// TwinCAT 3 PLC project LSS_LIB
// Title: LSS
// Company: SLAC
// ProjectVersion: 0.0.0
// ProgramVersion: 3.1.4026.17
// libraries:
//   Tc2_SerialCom, * (Beckhoff Automation GmbH)
//   Tc2_Standard, * (Beckhoff Automation GmbH)
//   Tc2_System, * (Beckhoff Automation GmbH)
//   Tc2_Utilities, * (Beckhoff Automation GmbH)
// project tree:
//   DUTs/ E_ALPHA_LED_LINE_POSITION.TcDUT, E_ALPHA_MULTIPLEX_ITEM.TcDUT
//   / PlcTask.TcTTO
//   POUs/ FB_Alpha215C.TcPOU, FB_ALPHA215C_Multiplex.TcPOU, MAIN.TcPOU
// real-time tasks:
//   TASK PlcTask: cycle T#10ms, priority 20, ADS port 350

CONFIGURATION LSS_LIB
    RESOURCE PLC ON TwinCAT3
        TASK PlcTask(INTERVAL := T#10ms, PRIORITY := 20);
        PROGRAM MAIN WITH PlcTask : MAIN;
    END_RESOURCE
END_CONFIGURATION

// ---- DUTs/E_ALPHA_LED_LINE_POSITION.TcDUT
{attribute 'qualified_only'}
{attribute 'strict'}
{attribute 'to_string'}
TYPE E_ALPHA_LED_LINE_POSITION :
(
    MIDDLE_LINE := 0 	// — Text centered vertically
    (*
    TOP_LINE, 			(*— Text begins on the top line of the sign and the sign will use all its lines minus 1 in order
                        to display the text. For example, a 6-line sign will allow a maximum of 5 lines (6 minus 1) for the Top
                        Position. The Top/Bottom Line break will remain fixed until the next Middle or Fill position is
                        specified*)
    BOTTOM_LINE, 		(* — The starting position of the Bottom Line(s) immediately follows the last line of the
                        Top Line. For example, a 6-line sign with 3 lines of text associated with the Top Line would start the
                        Bottom Line text on the 4th line of the sign. *)

    FILL				(*he sign will fill all available lines, centering the lines vertically*)
    *)
);
END_TYPE

// ---- DUTs/E_ALPHA_MULTIPLEX_ITEM.TcDUT
TYPE E_ALPHA_MULTIPLEX_ITEM :
STRUCT
    sMessage : STRING := ' ';
    sAddress : STRING := '00'; // Display on all signs. Or Specific
    sFile	: STRING := '0'; // Sign Default configuration file 1; file 0 is priotiry
    tTime : TIME := T#1S; // How long message should display
    bActive : BOOL := FALSE; // Message should be displayed.
END_STRUCT
END_TYPE

// ---- POUs/MAIN.TcPOU
PROGRAM MAIN
VAR
END_VAR

END_PROGRAM

// ---- POUs/FB_Alpha215C.TcPOU
FUNCTION_BLOCK FB_Alpha215C
(*This FB can be used to send print commands to the ALpha Signs*)
VAR_INPUT
END_VAR
VAR_OUTPUT
END_VAR
VAR
	fbBackgroundSerialLine: SerialLineControl;
	RxBuffer:   ComBuffer;
    TxBuffer:   ComBuffer;

	// Link to hardware.
	stComIn		AT %I*	:	EL6inData22B (*KL6inData22B*);
    stComOut	AT %Q*	:	EL6outData22B (*KL6outData22B*);

	//sCommand : STRING := '';  // (sCommand = sCommandCode + sDataField) + sCommand // NESTING commands
	//sSendMessage : STRING := '_00_00_00_00_00_01Z00_02A0_1Ba_1A9_1C1NO ACCESS_04';

	bBackgroundComError: BOOL;
	bBackgroundErrorId: UINT;
	bBackgroundTaskRunning : BOOL;

	fbClearComBuffer		: ClearComBuffer;
    fbSendString			: SendString;
    fbReceiveString			: ReceiveString;

	sSendPacket : STRING := '';

	bExecuteSend : BOOL := FALSE;
	iState : UINT := 0;

	fbRingBuff : FB_StringRingBuffer;
	fbBufferMemory    : ARRAY[0..2048] OF BYTE;
	
	tTimer : TON;

END_VAR

fbRingBuff(pBuffer := ADR(fbBufferMemory), cbBuffer := SIZEOF(fbBufferMemory));
tTimer(IN:=TRUE, PT:= T#100MS);

CASE iState OF
	0:
		IF bExecuteSend THEN // Manual Send
			fbSendString.SendString := sSendPacket;
			fbClearComBuffer(Buffer:=TxBuffer);
			iState := 10;
		END_IF

		IF fbRingBuff.nCount > 0 THEN // Send w/ ring buffer
			fbRingBuff.A_RemoveHead();
			sSendPacket := fbRingBuff.getValue;
			fbSendString.SendString := sSendPacket;
			fbClearComBuffer(Buffer:=TxBuffer);
			iState := 10;
		END_IF

	10: // SEND PACKET

		fbSendString(TXbuffer:=TxBuffer);

		IF NOT fbSendString.Busy AND fbSendString.Error = 0 THEN
			tTimer.IN := FALSE;
			tTimer();
			iState := 20;
		END_IF
		
	20: // WAIT FOR NEXT MESSAGE TO SEND
		IF tTimer.Q THEN
			bExecuteSend := FALSE;
			sSendPacket := '';
			iState := 0;
		END_IF

END_CASE

ACTION A_RUN_BACKGROUND_SERIAL_CONTROL:

bBackgroundTaskRunning := TRUE;

fbBackgroundSerialLine(
	Mode := ComSerialLineMode_t.SERIALLINEMODE_EL6_22B,
	pComIn := ADR(stComIn),
	pComOut := ADR(stComout),
	SizeComIn:= UINT_TO_INT(SIZEOF(stComout)),
    TxBuffer:= TxBuffer,
    RxBuffer:= RxBuffer,
	Error => bBackgroundComError,
	ErrorID => bBackgroundErrorId);
END_ACTION

METHOD PRIVATE M_BUILD_PACKET : STRING
VAR_INPUT
	sCommand : STRING;
	sAddress : STRING;
END_VAR
VAR
	sPacket : STRING := '';
	// TRANSMISSION FORMAT: <NULL> <SOH> <TypeCode> <SignAdress> <STX> <CommandCode> <DataField> <EOT>

	NULL : STRING := '_00_00_00_00_00';	(*A minimum of five <NUL>s (00H) must be transmitted as packet synchronization characters.
											 Five <SOH>s (01H) may be substituted for the five <NUL>s.
											 The sign uses these five characters to establish the baud rate *)

	SOH : STRING := '_01';	// Start of Header
	TYPE_CODE : STRING := 'Z';	// Set Type of Sign; 'Z' = All signs
	STX : STRING :='_02'; 		//“Start of TeXt” (02H) character. <STX> always precedes a Command Code.
	EOT : STRING:= '_04';		// "End of Transmission'
END_VAR
sPacket := CONCAT(sPacket, NULL);
sPacket := CONCAT(sPacket, SOH);
sPacket := CONCAT(sPacket, TYPE_CODE);
sPacket := CONCAT(sPacket, sAddress);
sPacket := CONCAT(sPacket, STX);
sPacket := CONCAT(sPacket, sCommand);
sPacket := CONCAT(sPacket, EOT);

M_BUILD_PACKET := sPacket;
END_METHOD

METHOD PRIVATE M_BUILD_TEXT_WRITE_COMMAND : STRING
VAR_INPUT
	sMessage : STRING;
	iFile : STRING := '0'; // print to priotiry file; so message shows up immediatly
	eLinePos : E_ALPHA_LED_LINE_POSITION := E_ALPHA_LED_LINE_POSITION.MIDDLE_LINE;

END_VAR
VAR
	COMMAND_CODE : STRING := 'A'; // A = WRITE TO 'FILE'
	ESC : STRING := '_1B';
	LINE_POS : STRING;
	MODE_CODE : STRING := 'b_1C1'; // func that chains multiple codes? ; Holds Text in place (b); red color text (_1C1) - this can chain multiple codes.
	SPECIAL_MODE : STRING := ''; // CAN ALSO BE ENUM
	// A - WRITE
	// 0 - FILE LABEL ;0 is Prority
	// _1B - ESCAPE CHAR
	// '' - LINE POSITION
	// a - MODE CODE
	// '' - SPECIAL MODE
	// _1A9_1C1NO ACCESS - TEXT

	sCommand : STRING;
END_VAR
CASE eLinePos OF
	E_ALPHA_LED_LINE_POSITION.MIDDLE_LINE:
		LINE_POS := ' ';
END_CASE

sCommand := CONCAT(sCommand, COMMAND_CODE);
sCommand := CONCAT(sCommand, iFile);
sCommand := CONCAT(sCommand, ESC);
sCommand := CONCAT(sCommand, LINE_POS);
sCommand := CONCAT(sCommand, MODE_CODE);
sCommand := CONCAT(sCommand, SPECIAL_MODE);
sCommand := CONCAT(sCommand, sMessage);

M_BUILD_TEXT_WRITE_COMMAND := sCommand;
END_METHOD

METHOD M_Print : BOOL
VAR_INPUT
	sAddress : STRING := '00'; // default broadcast to all
	iFile : STRING := '0'; // Use Priority file to instantly send message to sign.
	sMessage : STRING;
END_VAR
VAR
	sCommand : STRING;
	sPacket : STRING;
END_VAR
sCommand := M_BUILD_TEXT_WRITE_COMMAND(sMessage, iFile);
sPacket := M_BUILD_PACKET(sCommand, sAddress);

fbRingBuff.putValue := sPacket;
fbRingBuff.A_AddTail();
END_METHOD

END_FUNCTION_BLOCK

// ---- POUs/FB_ALPHA215C_Multiplex.TcPOU
FUNCTION_BLOCK FB_ALPHA215C_Multiplex
(*This FB Add Messages to sign and cycle though multiple messages. Idealy One FB per Sign.
Otherwise some messages will display longer in some signs.

st_message
- message 	(string)
- duration	(time)

*)
VAR_INPUT
END_VAR
VAR_IN_OUT
    aMessages : ARRAY [*] OF E_ALPHA_MULTIPLEX_ITEM;
    aAlphaDriver : FB_Alpha215C;
END_VAR
VAR
    iCurrentItem : DINT :=  LOWER_BOUND(aMessages,1);
    iMultiplexState : UINT := 10;
    tTimer : TON;
    stItem : E_ALPHA_MULTIPLEX_ITEM;

END_VAR

tTimer(IN:=TRUE);

CASE iMultiplexState OF
    10: // START PRINTING
        stItem := aMessages[iCurrentItem];

        IF stItem.bActive THEN
            aAlphaDriver.M_Print(sAddress := stItem.sAddress,
                iFile := stItem.sFile,
                sMessage := stItem.sMessage
            );

            tTimer.PT := stItem.tTime;
        ELSE
            tTimer.PT := T#0S;
        END_IF

        tTimer.IN := FALSE; // START TIMER
        tTimer();
        iMultiplexState := 20;

    20: // Wait
        IF tTimer.Q THEN //
            iCurrentItem := iCurrentItem + 1;

            IF iCurrentItem > UPPER_BOUND(aMessages, 1) THEN
                iCurrentItem := LOWER_BOUND(aMessages,1);
            END_IF
            iMultiplexState := 10;
        END_IF

END_CASE

END_FUNCTION_BLOCK
